TEXTLIST E_DeformationType
  0 = 'NoDeformation'
  1 = 'ScriptGrid'
  2 = 'ScriptGridTrend'
  3 = 'LocalMarks1D'
   = ''
END_TEXTLIST

(* stored: Version 1.1.0.1, ProductVersion 3.1.4024.11
   TextList E_DeformationType: Id {f621b1d4-a856-40b7-8dcb-35e17927c651} *)
